# EPICS substitutions: ecmcApp/Db/SlitX-xr-extra.substitutions
file "ecmc-extra.template"
{
pattern
{P,      M,    R,   PORT, ADDR, PREC, HOMEPROC}
{IOC2:,  xr, xr-,   MCU1, 4,    3,    3}
}
